// TIA Portal V16 export
// export: Created 2021-11-12T13:31:27.6202778Z, ExportSetting WithDefaults, DisplayName Totally Integrated Automation Portal, DisplayVersion V16 Update 3, DisplayName TIA Portal Version Control Interface, DisplayVersion V16 Update 2, DisplayName TIA Portal Openness, DisplayVersion V16 Update 3, DisplayName SINAMICS Startdrive Advanced, DisplayVersion V16 Update 5, DisplayName SINAMICS Startdrive G130, G150, S120, S150, SINAMICS MV, S210, DisplayVersion V16 Update 5, DisplayName SINAMICS Startdrive G110M, G120, G120C, G120D, G120P, G115D, DisplayVersion V16 Update 5, DisplayName STEP 7 Professional, DisplayVersion V16 Update 3, DisplayName STEP 7 Safety, DisplayVersion V16, DisplayName WinCC UA Professional, DisplayVersion V16 Update 3
FUNCTION_BLOCK "STD_PartCounter"   // FB50, LAD
{ S7_Optimized_Access := 'TRUE' }
VERSION : 0.1
// MICE standard block 
// PartCounter
// Block counts parts
// 
// 
// Version              Created                        by             Comment
// 0.1                      18.6. 2019                   MSt           initial version
// stored: AutoNumber true, IsIECCheckEnabled false, IsRetainMemResEnabled false, MemoryReserve 100, SetENOAutomatically false, UDAEnableTagReadback false
   VAR_INPUT
      IB1CountPulse : Bool;   // Signal of incomming part(s)
      IB1NegEdge : Bool;   // Count on negative edge
      ID_NoOfPartsOnPulse : DInt;   // Number of parts added by one pulse
      IB1ResetCounter : Bool;   // Clear counter
      IB1SetCounter : Bool;   // Set couter to defined value
      ID_SetValue : DInt;   // Value that will be set by IB1SetCounter
      IB1Ack : Bool;   // Alarm reset
      IB1AlarmSuppress : Bool;   // Alarm suppression
   END_VAR
   VAR_OUTPUT
      OS_Status : Struct   // Output signal
         Main : "UDT_Status_main";
         Specific : "UDT_PartCounter_Status";
         Error : "UDT_Error01";
      END_STRUCT;
      ODIValue : DInt;   // Value of counter
      OB1Full : Bool;   // Number of part > defined value for BinFull
   END_VAR
   VAR_IN_OUT
      XS_Parameter : "UDT_PartCounter_Parameter";
      XS_Command : "UDT_PartCounter_Command";
   END_VAR
   VAR
      SS_Alarm { ExternalAccessible := 'False'; ExternalVisible := 'False'; ExternalWritable := 'False'} : Struct   // Device alarms
         Overloaded { ExternalAccessible := 'False'; ExternalVisible := 'False'; ExternalWritable := 'False'} : Bool;   // Alarm / Alarme
         Res_0_1 { ExternalAccessible := 'False'; ExternalVisible := 'False'; ExternalWritable := 'False'} : Bool;   // Fail / Porucha / La panne
         Res_0_2 { ExternalAccessible := 'False'; ExternalVisible := 'False'; ExternalWritable := 'False'} : Bool;
         Res_0_3 { ExternalAccessible := 'False'; ExternalVisible := 'False'; ExternalWritable := 'False'} : Bool;
         Res_0_4 { ExternalAccessible := 'False'; ExternalVisible := 'False'; ExternalWritable := 'False'} : Bool;
         Res_0_5 { ExternalAccessible := 'False'; ExternalVisible := 'False'; ExternalWritable := 'False'} : Bool;
         Res_0_6 { ExternalAccessible := 'False'; ExternalVisible := 'False'; ExternalWritable := 'False'} : Bool;
         Res_0_7 { ExternalAccessible := 'False'; ExternalVisible := 'False'; ExternalWritable := 'False'} : Bool;
         Res_1_0 { ExternalAccessible := 'False'; ExternalVisible := 'False'; ExternalWritable := 'False'} : Bool;
         Res_1_1 { ExternalAccessible := 'False'; ExternalVisible := 'False'; ExternalWritable := 'False'} : Bool;
         Res_1_2 { ExternalAccessible := 'False'; ExternalVisible := 'False'; ExternalWritable := 'False'} : Bool;
         Res_1_3 { ExternalAccessible := 'False'; ExternalVisible := 'False'; ExternalWritable := 'False'} : Bool;
         Res_1_4 { ExternalAccessible := 'False'; ExternalVisible := 'False'; ExternalWritable := 'False'} : Bool;
         Res_1_5 { ExternalAccessible := 'False'; ExternalVisible := 'False'; ExternalWritable := 'False'} : Bool;
         Res_1_6 { ExternalAccessible := 'False'; ExternalVisible := 'False'; ExternalWritable := 'False'} : Bool;
         Res_1_7 { ExternalAccessible := 'False'; ExternalVisible := 'False'; ExternalWritable := 'False'} : Bool;
      END_STRUCT;
      SS_Warning { ExternalAccessible := 'False'; ExternalVisible := 'False'; ExternalWritable := 'False'} : Struct   // Device warnings
         TooManyParts { ExternalAccessible := 'False'; ExternalVisible := 'False'; ExternalWritable := 'False'} : Bool;   // A lot of parts in bin / Varování / Avertissement
         Res_0_1 { ExternalAccessible := 'False'; ExternalVisible := 'False'; ExternalWritable := 'False'} : Bool;   // Tolerance / Tolérance
         Res_0_2 { ExternalAccessible := 'False'; ExternalVisible := 'False'; ExternalWritable := 'False'} : Bool;   // Operátorská zpráva / Le rapport de l ’ utilisateur
         Res_0_3 { ExternalAccessible := 'False'; ExternalVisible := 'False'; ExternalWritable := 'False'} : Bool;
         Res_0_4 { ExternalAccessible := 'False'; ExternalVisible := 'False'; ExternalWritable := 'False'} : Bool;
         Res_0_5 { ExternalAccessible := 'False'; ExternalVisible := 'False'; ExternalWritable := 'False'} : Bool;
         Res_0_6 { ExternalAccessible := 'False'; ExternalVisible := 'False'; ExternalWritable := 'False'} : Bool;
         Res_0_7 { ExternalAccessible := 'False'; ExternalVisible := 'False'; ExternalWritable := 'False'} : Bool;
         Res_1_0 { ExternalAccessible := 'False'; ExternalVisible := 'False'; ExternalWritable := 'False'} : Bool;
         Res_1_1 { ExternalAccessible := 'False'; ExternalVisible := 'False'; ExternalWritable := 'False'} : Bool;
         Res_1_2 { ExternalAccessible := 'False'; ExternalVisible := 'False'; ExternalWritable := 'False'} : Bool;
         Res_1_3 { ExternalAccessible := 'False'; ExternalVisible := 'False'; ExternalWritable := 'False'} : Bool;
         Res_1_4 { ExternalAccessible := 'False'; ExternalVisible := 'False'; ExternalWritable := 'False'} : Bool;
         Res_1_5 { ExternalAccessible := 'False'; ExternalVisible := 'False'; ExternalWritable := 'False'} : Bool;
         Res_1_6 { ExternalAccessible := 'False'; ExternalVisible := 'False'; ExternalWritable := 'False'} : Bool;
         Res_1_7 { ExternalAccessible := 'False'; ExternalVisible := 'False'; ExternalWritable := 'False'} : Bool;
      END_STRUCT;
      SS_Edge : Array[0..15] of Bool;
      SB1IsEmpty : Bool;
      SB1IsFull : Bool;
   END_VAR
   VAR RETAIN
      SDICounter : DInt;   // Value of counter
   END_VAR
   VAR_TEMP
      TS_Parameter : "UDT_PartCounter_Parameter";   // Parameters to/from HMI
      TS_Command : "UDT_PartCounter_Command";   // Commands from HMI
      TS_Status : Struct   // Output signal
         Main : "UDT_Status_main";
         Specific : "UDT_PartCounter_Status";
         Error : "UDT_Error01";
      END_STRUCT;
   END_VAR
   VAR_TEMP   // added for the SCL form of the ladder/FBD networks
      _w1 : Bool;
      _w2 : Bool;
   END_VAR
BEGIN

REGION Network 1: Clear temporary variables
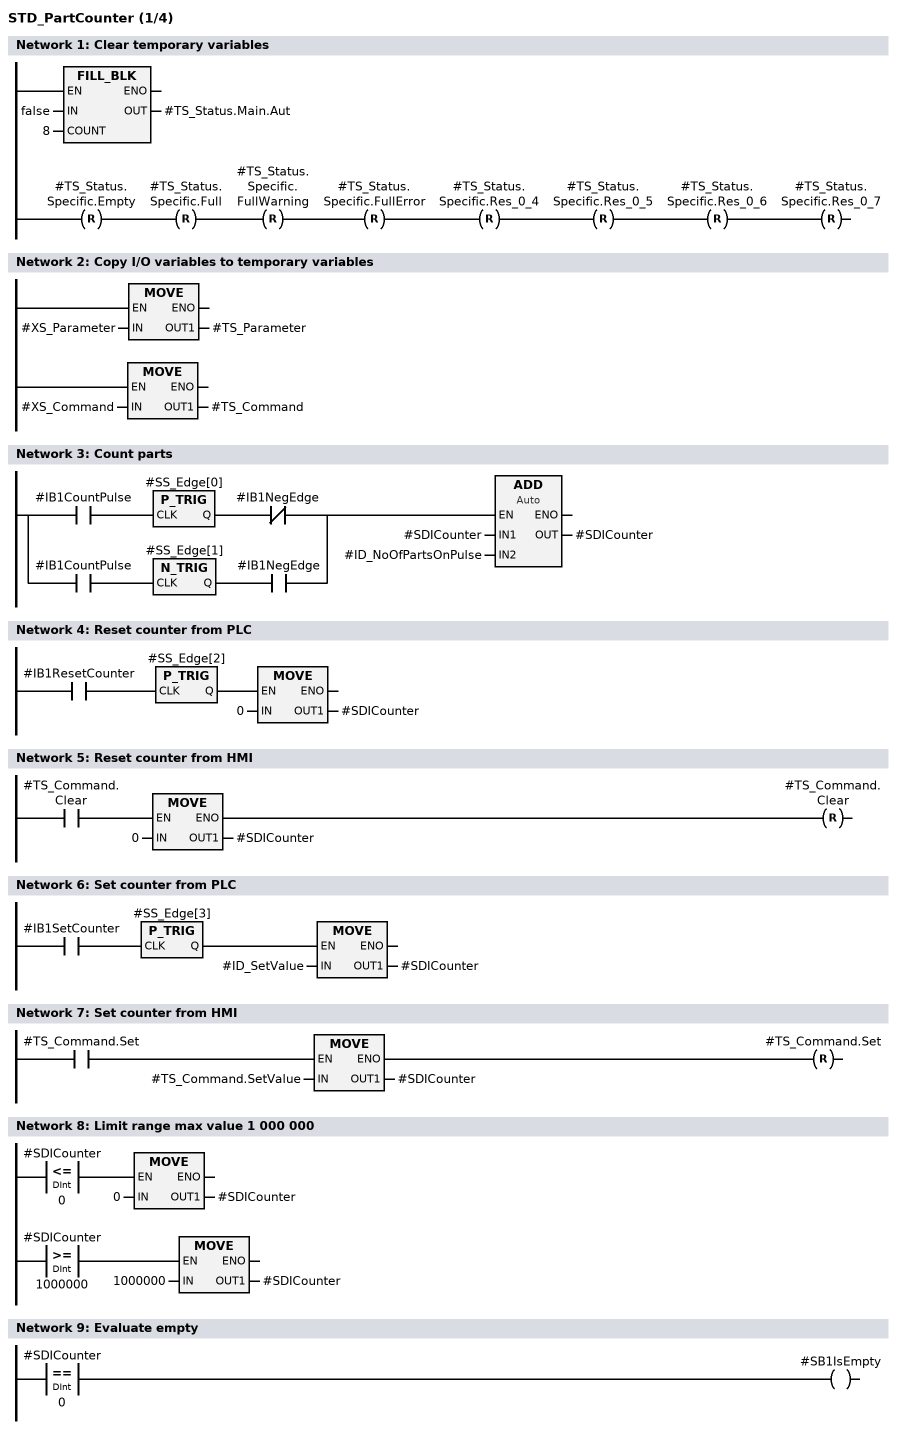
   RUNG wire#powerrail
      FillBlockI(in := false, count := 8, out => #TS_Status.Main.Aut)
   END_RUNG
   RUNG wire#powerrail
      R_Coil( #TS_Status.Specific.Empty )
      R_Coil( #TS_Status.Specific.Full )
      R_Coil( #TS_Status.Specific.FullWarning )
      R_Coil( #TS_Status.Specific.FullError )
      R_Coil( #TS_Status.Specific.Res_0_4 )
      R_Coil( #TS_Status.Specific.Res_0_5 )
      R_Coil( #TS_Status.Specific.Res_0_6 )
      R_Coil( #TS_Status.Specific.Res_0_7 )
   END_RUNG
   // the same network as SCL:
   FILL_BLK(IN := false, COUNT := 8, OUT => #TS_Status.Main.Aut);
   #TS_Status.Specific.Empty := FALSE;
   #TS_Status.Specific.Full := FALSE;
   #TS_Status.Specific.FullWarning := FALSE;
   #TS_Status.Specific.FullError := FALSE;
   #TS_Status.Specific.Res_0_4 := FALSE;
   #TS_Status.Specific.Res_0_5 := FALSE;
   #TS_Status.Specific.Res_0_6 := FALSE;
   #TS_Status.Specific.Res_0_7 := FALSE;
END_REGION

REGION Network 2: Copy I/O variables to temporary variables
   RUNG wire#powerrail
      { S7_GenerateENO := "TRUE" } Move(in := #XS_Parameter, out1 => #TS_Parameter)
   END_RUNG
   RUNG wire#powerrail
      { S7_GenerateENO := "TRUE" } Move(in := #XS_Command, out1 => #TS_Command)
   END_RUNG
   // the same network as SCL:
   #TS_Parameter := #XS_Parameter;
   #TS_Command := #XS_Command;
END_REGION

REGION Network 3: Count parts
   RUNG wire#powerrail
      Contact( #IB1CountPulse )
      P_Trig( #SS_Edge[0] )
      I_Contact( #IB1NegEdge )
      wire#w1
      Add(in1 := #SDICounter, in2 := #ID_NoOfPartsOnPulse, out => #SDICounter)
   END_RUNG
   RUNG wire#powerrail
      Contact( #IB1CountPulse )
      N_Trig( #SS_Edge[1] )
      Contact( #IB1NegEdge )
   END_RUNG wire#w1
   // the same network as SCL:
   #_w1 := #IB1CountPulse AND NOT #SS_Edge[0];   // rising edge
   #SS_Edge[0] := #IB1CountPulse;
   #_w2 := NOT #IB1CountPulse AND #SS_Edge[1];   // falling edge
   #SS_Edge[1] := #IB1CountPulse;
   IF (#_w1 AND NOT #IB1NegEdge) OR (#_w2 AND #IB1NegEdge) THEN
       #SDICounter := #SDICounter + #ID_NoOfPartsOnPulse;
   END_IF;
END_REGION

REGION Network 4: Reset counter from PLC
   RUNG wire#powerrail
      Contact( #IB1ResetCounter )
      P_Trig( #SS_Edge[2] )
      Move(in := 0, out1 => #SDICounter)
   END_RUNG
   // the same network as SCL:
   #_w1 := #IB1ResetCounter AND NOT #SS_Edge[2];   // rising edge
   #SS_Edge[2] := #IB1ResetCounter;
   IF #_w1 THEN #SDICounter := 0; END_IF;
END_REGION

REGION Network 5: Reset counter from HMI
   RUNG wire#powerrail
      Contact( #TS_Command.Clear )
      Move(in := 0, out1 => #SDICounter)
      R_Coil( #TS_Command.Clear )
   END_RUNG
   // the same network as SCL:
   IF #TS_Command.Clear THEN
       #SDICounter := 0;
       #TS_Command.Clear := FALSE;
   END_IF;
END_REGION

REGION Network 6: Set counter from PLC
   RUNG wire#powerrail
      Contact( #IB1SetCounter )
      P_Trig( #SS_Edge[3] )
      Move(in := #ID_SetValue, out1 => #SDICounter)
   END_RUNG
   // the same network as SCL:
   #_w1 := #IB1SetCounter AND NOT #SS_Edge[3];   // rising edge
   #SS_Edge[3] := #IB1SetCounter;
   IF #_w1 THEN #SDICounter := #ID_SetValue; END_IF;
END_REGION

REGION Network 7: Set counter from HMI
   RUNG wire#powerrail
      Contact( #TS_Command.Set )
      Move(in := #TS_Command.SetValue, out1 => #SDICounter)
      R_Coil( #TS_Command.Set )
   END_RUNG
   // the same network as SCL:
   IF #TS_Command.Set THEN
       #SDICounter := #TS_Command.SetValue;
       #TS_Command.Set := FALSE;
   END_IF;
END_REGION

REGION Network 8: Limit range max value 1 000 000
   RUNG wire#powerrail
      { S7_Templates := "SrcType := DInt" } LE_Contact(in1 := #SDICounter, in2 := 0)
      Move(in := 0, out1 => #SDICounter)
   END_RUNG
   RUNG wire#powerrail
      { S7_Templates := "SrcType := DInt" } GE_Contact(in1 := #SDICounter, in2 := 1000000)
      Move(in := 1000000, out1 => #SDICounter)
   END_RUNG
   // the same network as SCL:
   IF #SDICounter <= 0 THEN #SDICounter := 0; END_IF;
   IF #SDICounter >= 1000000 THEN #SDICounter := 1000000; END_IF;
END_REGION

REGION Network 9: Evaluate empty
   RUNG wire#powerrail
      { S7_Templates := "SrcType := DInt" } EQ_Contact(in1 := #SDICounter, in2 := 0)
      Coil( #SB1IsEmpty )
   END_RUNG
   // the same network as SCL:
   #SB1IsEmpty := #SDICounter = 0;
END_REGION

REGION Network 10: Evaluate full
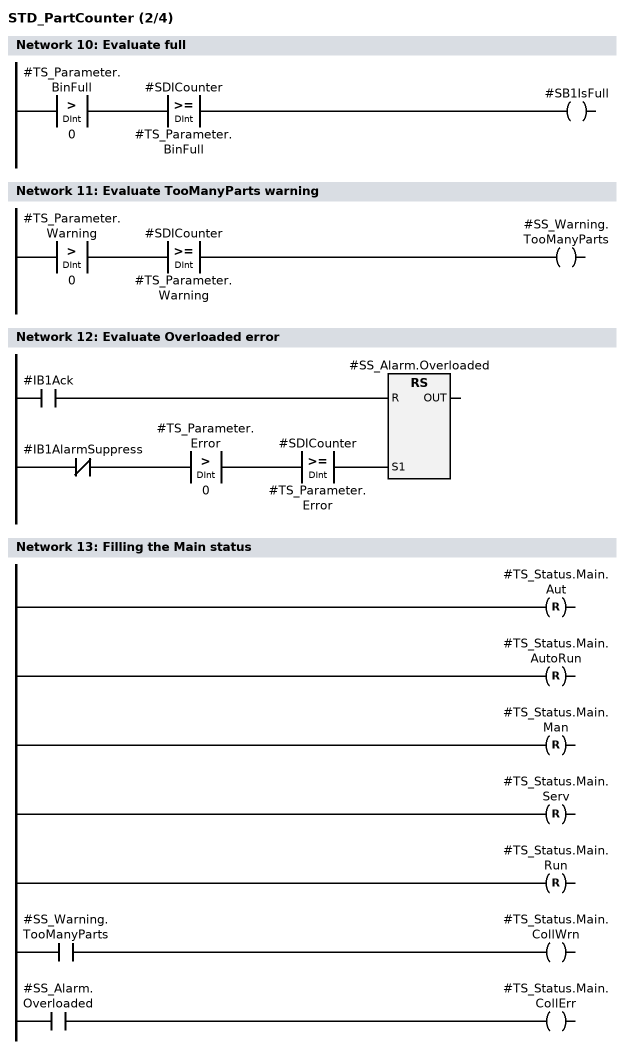
   RUNG wire#powerrail
      { S7_Templates := "SrcType := DInt" } GT_Contact(in1 := #TS_Parameter.BinFull, in2 := 0)
      { S7_Templates := "SrcType := DInt" } GE_Contact(in1 := #SDICounter, in2 := #TS_Parameter.BinFull)
      Coil( #SB1IsFull )
   END_RUNG
   // the same network as SCL:
   #SB1IsFull := (#TS_Parameter.BinFull > 0) AND (#SDICounter >= #TS_Parameter.BinFull);
END_REGION

REGION Network 11: Evaluate TooManyParts warning
   RUNG wire#powerrail
      { S7_Templates := "SrcType := DInt" } GT_Contact(in1 := #TS_Parameter.Warning, in2 := 0)
      { S7_Templates := "SrcType := DInt" } GE_Contact(in1 := #SDICounter, in2 := #TS_Parameter.Warning)
      Coil( #SS_Warning.TooManyParts )
   END_RUNG
   // the same network as SCL:
   #SS_Warning.TooManyParts := (#TS_Parameter.Warning > 0) AND (#SDICounter >= #TS_Parameter.Warning);
END_REGION

REGION Network 12: Evaluate Overloaded error
   RUNG wire#powerrail
      Contact( #IB1Ack )
      S_RS(operand := #SS_Alarm.Overloaded, s1 := wire#w1)
   END_RUNG
   RUNG wire#powerrail
      I_Contact( #IB1AlarmSuppress )
      { S7_Templates := "SrcType := DInt" } GT_Contact(in1 := #TS_Parameter.Error, in2 := 0)
      { S7_Templates := "SrcType := DInt" } GE_Contact(in1 := #SDICounter, in2 := #TS_Parameter.Error)
   END_RUNG wire#w1
   // the same network as SCL:
   IF #IB1Ack THEN
       #SS_Alarm.Overloaded := FALSE;   // RS flip-flop
   END_IF;
   IF NOT #IB1AlarmSuppress AND (#TS_Parameter.Error > 0) AND (#SDICounter >= #TS_Parameter.Error) THEN
       #SS_Alarm.Overloaded := TRUE;
   END_IF;
END_REGION

REGION Network 13: Filling the Main status
   RUNG wire#powerrail
      R_Coil( #TS_Status.Main.Aut )
   END_RUNG
   RUNG wire#powerrail
      R_Coil( #TS_Status.Main.AutoRun )
   END_RUNG
   RUNG wire#powerrail
      R_Coil( #TS_Status.Main.Man )
   END_RUNG
   RUNG wire#powerrail
      R_Coil( #TS_Status.Main.Serv )
   END_RUNG
   RUNG wire#powerrail
      R_Coil( #TS_Status.Main.Run )
   END_RUNG
   RUNG wire#powerrail
      Contact( #SS_Warning.TooManyParts )
      Coil( #TS_Status.Main.CollWrn )
   END_RUNG
   RUNG wire#powerrail
      Contact( #SS_Alarm.Overloaded )
      Coil( #TS_Status.Main.CollErr )
   END_RUNG
   // the same network as SCL:
   #TS_Status.Main.Aut := FALSE;
   #TS_Status.Main.AutoRun := FALSE;
   #TS_Status.Main.Man := FALSE;
   #TS_Status.Main.Serv := FALSE;
   #TS_Status.Main.Run := FALSE;
   #TS_Status.Main.CollWrn := #SS_Warning.TooManyParts;
   #TS_Status.Main.CollErr := #SS_Alarm.Overloaded;
END_REGION

REGION Network 14: Filling the specific status
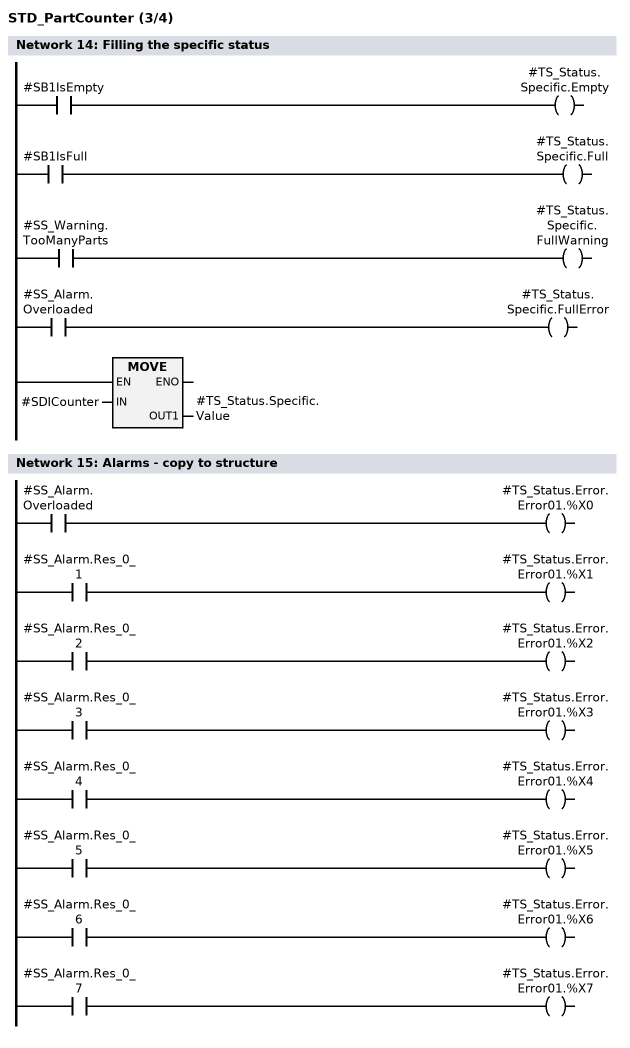
   RUNG wire#powerrail
      Contact( #SB1IsEmpty )
      Coil( #TS_Status.Specific.Empty )
   END_RUNG
   RUNG wire#powerrail
      Contact( #SB1IsFull )
      Coil( #TS_Status.Specific.Full )
   END_RUNG
   RUNG wire#powerrail
      Contact( #SS_Warning.TooManyParts )
      Coil( #TS_Status.Specific.FullWarning )
   END_RUNG
   RUNG wire#powerrail
      Contact( #SS_Alarm.Overloaded )
      Coil( #TS_Status.Specific.FullError )
   END_RUNG
   RUNG wire#powerrail
      Move(in := #SDICounter, out1 => #TS_Status.Specific.Value)
   END_RUNG
   // the same network as SCL:
   #TS_Status.Specific.Empty := #SB1IsEmpty;
   #TS_Status.Specific.Full := #SB1IsFull;
   #TS_Status.Specific.FullWarning := #SS_Warning.TooManyParts;
   #TS_Status.Specific.FullError := #SS_Alarm.Overloaded;
   #TS_Status.Specific.Value := #SDICounter;
END_REGION

REGION Network 15: Alarms - copy to structure
   RUNG wire#powerrail
      Contact( #SS_Alarm.Overloaded )
      Coil( #TS_Status.Error.Error01.%X0 )
   END_RUNG
   RUNG wire#powerrail
      Contact( #SS_Alarm.Res_0_1 )
      Coil( #TS_Status.Error.Error01.%X1 )
   END_RUNG
   RUNG wire#powerrail
      Contact( #SS_Alarm.Res_0_2 )
      Coil( #TS_Status.Error.Error01.%X2 )
   END_RUNG
   RUNG wire#powerrail
      Contact( #SS_Alarm.Res_0_3 )
      Coil( #TS_Status.Error.Error01.%X3 )
   END_RUNG
   RUNG wire#powerrail
      Contact( #SS_Alarm.Res_0_4 )
      Coil( #TS_Status.Error.Error01.%X4 )
   END_RUNG
   RUNG wire#powerrail
      Contact( #SS_Alarm.Res_0_5 )
      Coil( #TS_Status.Error.Error01.%X5 )
   END_RUNG
   RUNG wire#powerrail
      Contact( #SS_Alarm.Res_0_6 )
      Coil( #TS_Status.Error.Error01.%X6 )
   END_RUNG
   RUNG wire#powerrail
      Contact( #SS_Alarm.Res_0_7 )
      Coil( #TS_Status.Error.Error01.%X7 )
   END_RUNG
   // the same network as SCL:
   #TS_Status.Error.Error01.%X0 := #SS_Alarm.Overloaded;
   #TS_Status.Error.Error01.%X1 := #SS_Alarm.Res_0_1;
   #TS_Status.Error.Error01.%X2 := #SS_Alarm.Res_0_2;
   #TS_Status.Error.Error01.%X3 := #SS_Alarm.Res_0_3;
   #TS_Status.Error.Error01.%X4 := #SS_Alarm.Res_0_4;
   #TS_Status.Error.Error01.%X5 := #SS_Alarm.Res_0_5;
   #TS_Status.Error.Error01.%X6 := #SS_Alarm.Res_0_6;
   #TS_Status.Error.Error01.%X7 := #SS_Alarm.Res_0_7;
END_REGION

REGION Network 16: Warnings - copy to structure
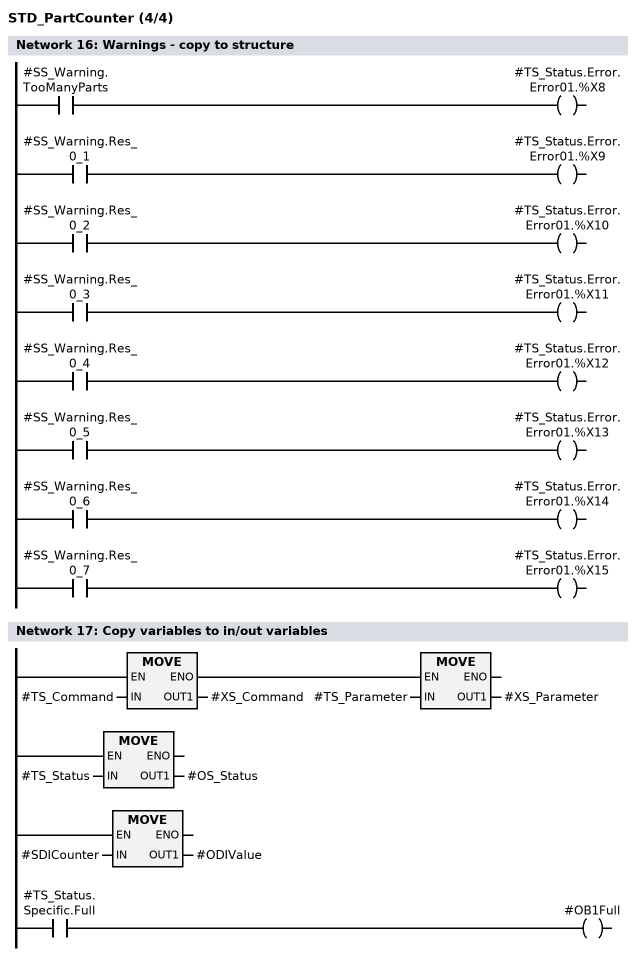
   RUNG wire#powerrail
      Contact( #SS_Warning.TooManyParts )
      Coil( #TS_Status.Error.Error01.%X8 )
   END_RUNG
   RUNG wire#powerrail
      Contact( #SS_Warning.Res_0_1 )
      Coil( #TS_Status.Error.Error01.%X9 )
   END_RUNG
   RUNG wire#powerrail
      Contact( #SS_Warning.Res_0_2 )
      Coil( #TS_Status.Error.Error01.%X10 )
   END_RUNG
   RUNG wire#powerrail
      Contact( #SS_Warning.Res_0_3 )
      Coil( #TS_Status.Error.Error01.%X11 )
   END_RUNG
   RUNG wire#powerrail
      Contact( #SS_Warning.Res_0_4 )
      Coil( #TS_Status.Error.Error01.%X12 )
   END_RUNG
   RUNG wire#powerrail
      Contact( #SS_Warning.Res_0_5 )
      Coil( #TS_Status.Error.Error01.%X13 )
   END_RUNG
   RUNG wire#powerrail
      Contact( #SS_Warning.Res_0_6 )
      Coil( #TS_Status.Error.Error01.%X14 )
   END_RUNG
   RUNG wire#powerrail
      Contact( #SS_Warning.Res_0_7 )
      Coil( #TS_Status.Error.Error01.%X15 )
   END_RUNG
   // the same network as SCL:
   #TS_Status.Error.Error01.%X8 := #SS_Warning.TooManyParts;
   #TS_Status.Error.Error01.%X9 := #SS_Warning.Res_0_1;
   #TS_Status.Error.Error01.%X10 := #SS_Warning.Res_0_2;
   #TS_Status.Error.Error01.%X11 := #SS_Warning.Res_0_3;
   #TS_Status.Error.Error01.%X12 := #SS_Warning.Res_0_4;
   #TS_Status.Error.Error01.%X13 := #SS_Warning.Res_0_5;
   #TS_Status.Error.Error01.%X14 := #SS_Warning.Res_0_6;
   #TS_Status.Error.Error01.%X15 := #SS_Warning.Res_0_7;
END_REGION

REGION Network 17: Copy variables to in/out variables
   RUNG wire#powerrail
      { S7_GenerateENO := "TRUE" } Move(in := #TS_Command, out1 => #XS_Command)
      { S7_GenerateENO := "TRUE" } Move(in := #TS_Parameter, out1 => #XS_Parameter)
   END_RUNG
   RUNG wire#powerrail
      { S7_GenerateENO := "TRUE" } Move(in := #TS_Status, out1 => #OS_Status)
   END_RUNG
   RUNG wire#powerrail
      Move(in := #SDICounter, out1 => #ODIValue)
   END_RUNG
   RUNG wire#powerrail
      Contact( #TS_Status.Specific.Full )
      Coil( #OB1Full )
   END_RUNG
   // the same network as SCL:
   // ENO of a box is taken as its EN; it also drops when the box reports an error
   #XS_Command := #TS_Command;
   #XS_Parameter := #TS_Parameter;
   #OS_Status := #TS_Status;
   #ODIValue := #SDICounter;
   #OB1Full := #TS_Status.Specific.Full;
END_REGION
END_FUNCTION_BLOCK
